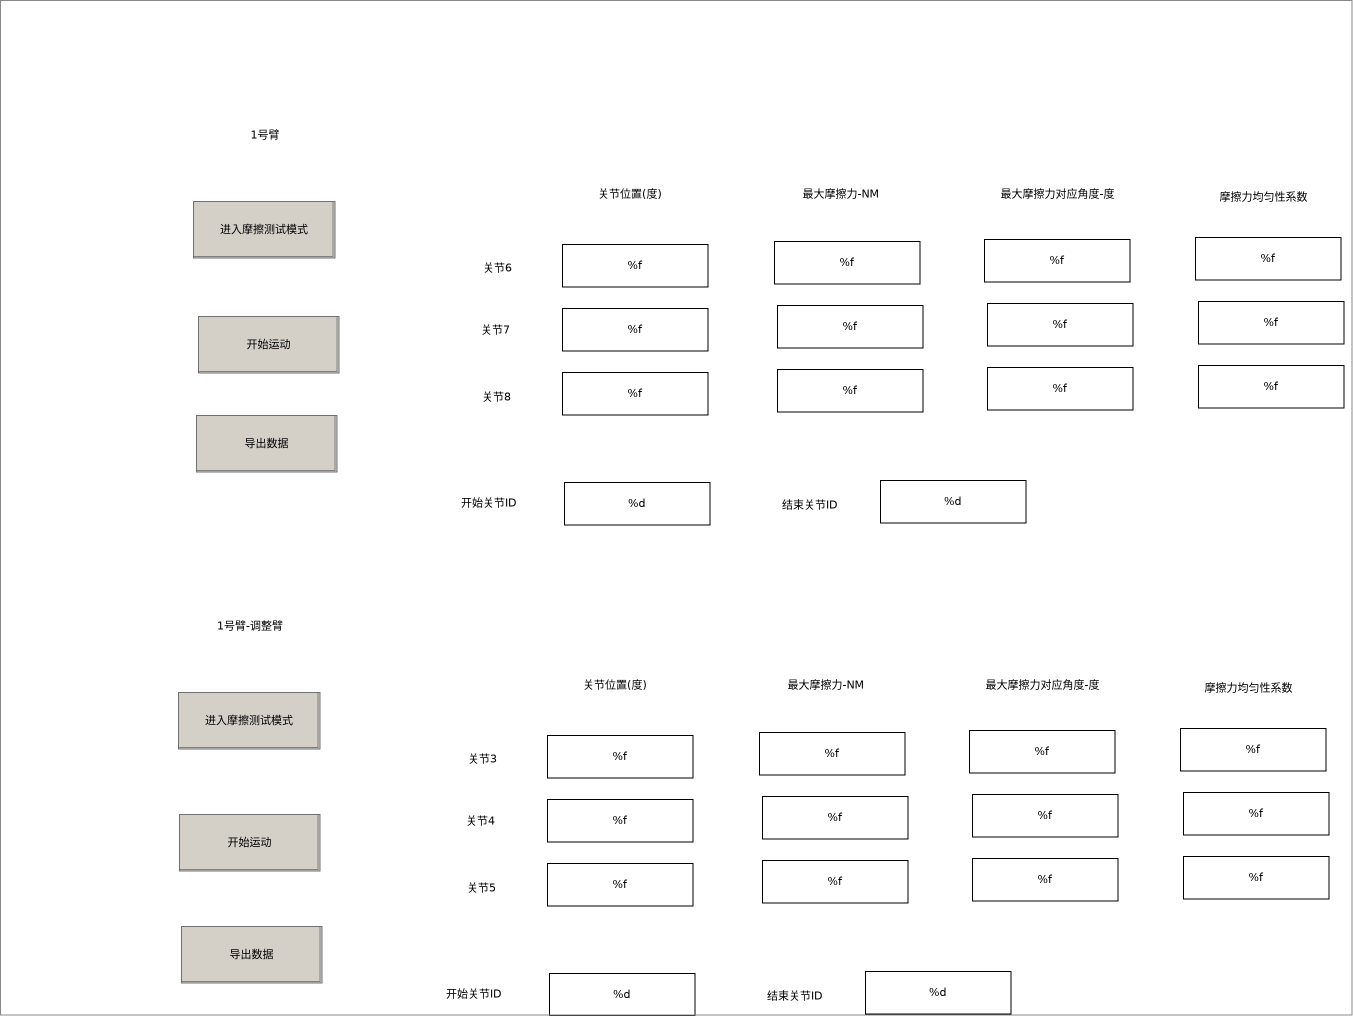
VISUALIZATION friction_a1  // 1353x1016
    Button (193,201 142x57), "进入摩擦测试模式", colour toggle: g_frictionTest.m_testMode[1]
        toggle g_frictionTest.m_testMode[1]
    Button (198,316 141x57), "开始运动", colour toggle: g_frictionTest.m_startMotion[1]
        toggle g_frictionTest.m_startMotion[1]
    Label (190,120 150x30), "1号臂"
    Rectangle (774,241 146x43), "%f", text variable: g_frictionTest.m_CoulombFrictionMax[1][1]
    Rectangle (777,305 146x43), "%f", text variable: g_frictionTest.m_CoulombFrictionMax[1][2]
    Rectangle (777,369 146x43), "%f", text variable: g_frictionTest.m_CoulombFrictionMax[1][3]
    Label (766,179 150x30), "最大摩擦力-NM"
    Rectangle (984,239 146x43), "%f", text variable: g_frictionTest.m_CoulombFrictionMax_JntPos[1][1]
    Rectangle (987,303 146x43), "%f", text variable: g_frictionTest.m_CoulombFrictionMax_JntPos[1][2]
    Rectangle (987,367 146x43), "%f", text variable: g_frictionTest.m_CoulombFrictionMax_JntPos[1][3]
    Label (941,179 233x30), "最大摩擦力对应角度-度"
    Rectangle (1195,237 146x43), "%f", text variable: g_frictionTest.m_CoulombFrictionRatio[1,1]
    Rectangle (1198,301 146x43), "%f", text variable: g_frictionTest.m_CoulombFrictionRatio[1,2]
    Rectangle (1198,365 146x43), "%f", text variable: g_frictionTest.m_CoulombFrictionRatio[1,3]
    Label (1174,182 179x30), "摩擦力均匀性系数"
    Rectangle (562,244 146x43), "%f", text variable: g_frictionTest.m_armDHJntPos[1][1]
    Label (446,250 103x36), "关节6"
    Label (444,312 103x36), "关节7"
    Label (445,379 103x36), "关节8"
    Rectangle (562,308 146x43), "%f", text variable: g_frictionTest.m_armDHJntPos[1][2]
    Rectangle (562,372 146x43), "%f", text variable: g_frictionTest.m_armDHJntPos[1][3]
    Label (555,179 150x30), "关节位置(度)"
    Label (414,488 150x30), "开始关节ID"
    Rectangle (564,482 146x43), "%d", text variable: g_frictionTest.m_jntIdStart[1]
        OnMouseClick: write the text variable via Default
    Label (735,490 150x30), "结束关节ID"
    Rectangle (880,480 146x43), "%d", text variable: g_frictionTest.m_jntIdEnd[1]
        OnMouseClick: write the text variable via Default
    Button (178,692 142x57), "进入摩擦测试模式", colour toggle: g_frictionTestSetup.m_testMode[1]
        toggle g_frictionTestSetup.m_testMode[1]
    Button (179,814 141x57), "开始运动", colour toggle: g_frictionTestSetup.m_startMotion[1]
        toggle g_frictionTestSetup.m_startMotion[1]
    Label (175,611 150x30), "1号臂-调整臂"
    Rectangle (759,732 146x43), "%f", text variable: g_frictionTestSetup.m_CoulombFrictionMax[1][3]
    Rectangle (762,796 146x43), "%f", text variable: g_frictionTestSetup.m_CoulombFrictionMax[1][4]
    Rectangle (762,860 146x43), "%f", text variable: g_frictionTestSetup.m_CoulombFrictionMax[1][5]
    Label (751,670 150x30), "最大摩擦力-NM"
    Rectangle (969,730 146x43), "%f", text variable: g_frictionTestSetup.m_CoulombFrictionMax_JntPos[1][3]
    Rectangle (972,794 146x43), "%f", text variable: g_frictionTestSetup.m_CoulombFrictionMax_JntPos[1][4]
    Rectangle (972,858 146x43), "%f", text variable: g_frictionTestSetup.m_CoulombFrictionMax_JntPos[1][5]
    Label (926,670 233x30), "最大摩擦力对应角度-度"
    Rectangle (1180,728 146x43), "%f", text variable: g_frictionTestSetup.m_CoulombFrictionRatio[1,3]
    Rectangle (1183,792 146x43), "%f", text variable: g_frictionTestSetup.m_CoulombFrictionRatio[1,4]
    Rectangle (1183,856 146x43), "%f", text variable: g_frictionTestSetup.m_CoulombFrictionRatio[1,5]
    Label (1159,673 179x30), "摩擦力均匀性系数"
    Rectangle (547,735 146x43), "%f", text variable: g_frictionTestSetup.m_armDHJntPos[1][3]
    Label (431,741 103x36), "关节3"
    Label (429,803 103x36), "关节4"
    Label (430,870 103x36), "关节5"
    Rectangle (547,799 146x43), "%f", text variable: g_frictionTestSetup.m_armDHJntPos[1][4]
    Rectangle (547,863 146x43), "%f", text variable: g_frictionTestSetup.m_armDHJntPos[1][5]
    Label (540,670 150x30), "关节位置(度)"
    Label (399,979 150x30), "开始关节ID"
    Rectangle (549,973 146x43), "%d", text variable: g_frictionTestSetup.m_jntIdStart[1]
        OnMouseClick: write the text variable via Default
    Label (720,981 150x30), "结束关节ID"
    Rectangle (865,971 146x43), "%d", text variable: g_frictionTestSetup.m_jntIdEnd[1]
        OnMouseClick: write the text variable via Default
    Button (196,415 141x57), "导出数据", colour toggle: g_frictionTest.m_duringWriteData[1]
        tap g_frictionTest.m_writeData[1]
    Button (181,926 141x57), "导出数据", colour toggle: g_frictionTestSetup.m_duringWriteData[1]
        tap g_frictionTestSetup.m_writeData[1]
END_VISUALIZATION

(* stored: Version 1.1.0.1, ProductVersion 3.1.4024.11
   Visu friction_a1: Id {5a775795-2dfc-41c7-a1ee-72e1b8a53633} *)
